TYPE ST_SystemParameter :
STRUCT
	Cylinder : ST_CylinderList;
	Servo : ST_ServoList;
	Mechanical : ST_MechanicalList;
	//Motor :ST_MotorList;
END_STRUCT
END_TYPE

(* stored: Version 1.1.0.1, ProductVersion 3.1.4024.13
   DUT ST_SystemParameter: Id {efb2311d-8ae5-4e25-925d-c45db23e9f11} *)
